PROGRAM MAIN
VAR
	udp1:  SampleUdpEchoServer;
END_VAR


udp1();

END_PROGRAM

(* stored: Version 1.1.0.1, ProductVersion 3.1.4024.16
   POU MAIN: Id {5ba6c13a-6ac1-4f7a-9948-296da78edcb1}, SpecialFunc None *)
